// SIMATIC S7-200 SMART project (STEP 7-Micro/WIN SMART), CPU SR40

ORGANIZATION_BLOCK 主程序:OB1
TITLE=程序注释
BEGIN
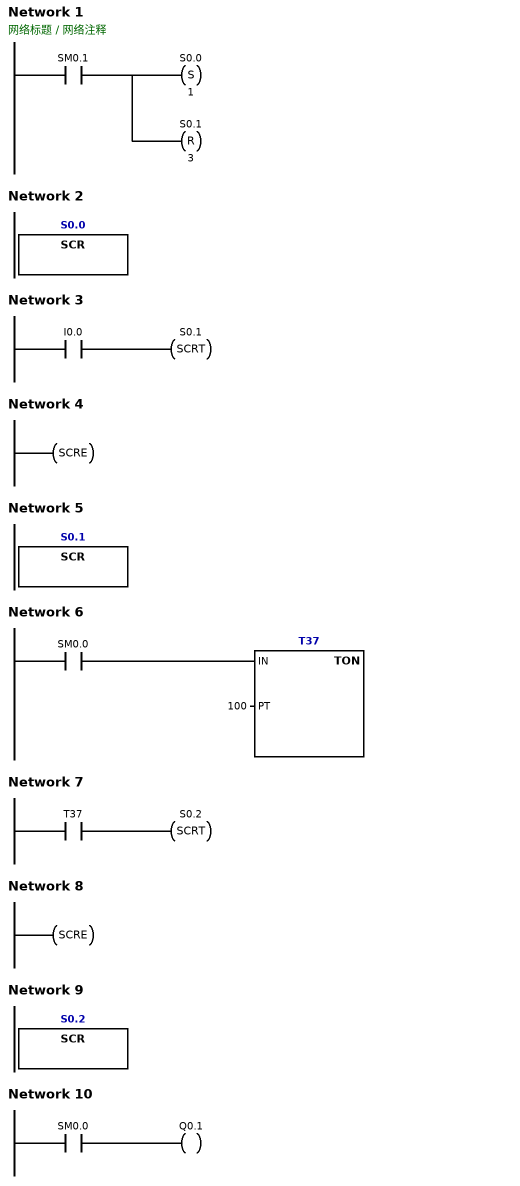
Network 1
// 网络标题
// 网络注释
LD     SM0.1
S      S0.0, 1
R      S0.1, 3
Network 2
LSCR   S0.0
Network 3
LD     I0.0
SCRT   S0.1
Network 4
SCRE
Network 5
LSCR   S0.1
Network 6
LD     SM0.0
TON    T37, 100
Network 7
LD     T37
SCRT   S0.2
Network 8
SCRE
Network 9
LSCR   S0.2
Network 10
LD     SM0.0
=      Q0.1
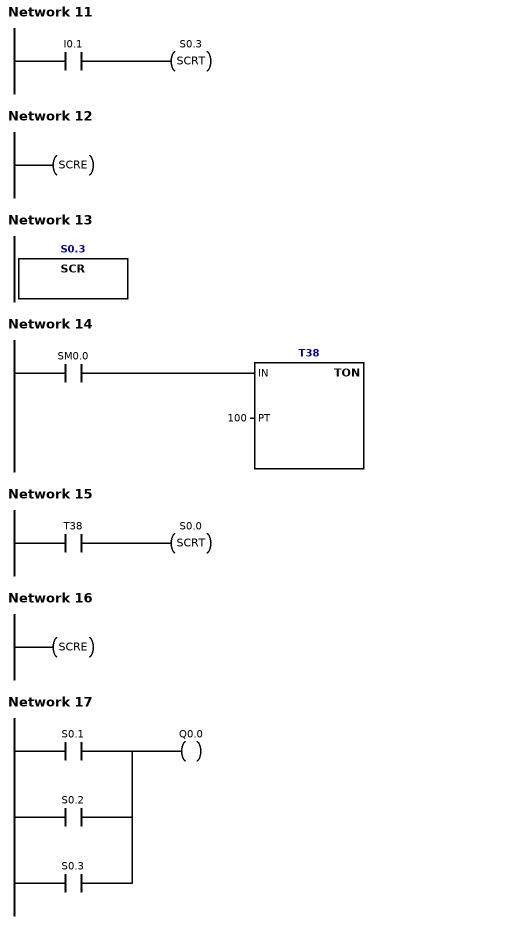
Network 11
LD     I0.1
SCRT   S0.3
Network 12
SCRE
Network 13
LSCR   S0.3
Network 14
LD     SM0.0
TON    T38, 100
Network 15
LD     T38
SCRT   S0.0
Network 16
SCRE
Network 17
LD     S0.1
O      S0.2
O      S0.3
=      Q0.0
END_ORGANIZATION_BLOCK
